(* IEC 61131-3 sources: AXOpen/src/components.zebra.vision/app/SystemConstants, 2 files *)

(* ---- plc_line_IoAddresses.st ---- *)
CONFIGURATION IoAddresses
    VAR_GLOBAL

        // Module EA3600/Data88Bin6Bout
        EA3600_Data88Bin6Bout_Input AT %IB0 : EA3600_Data88Bin6Bout_Input_Layout;
        EA3600_Data88Bin6Bout_Output AT %QB0 : EA3600_Data88Bin6Bout_Output_Layout;
    END_VAR
END_CONFIGURATION

TYPE
    EA3600_Data88Bin6Bout_Input_Layout : STRUCT
        Signals_0 AT %B0 : ARRAY[0..703] OF BOOL;
    END_STRUCT;
END_TYPE

TYPE
    EA3600_Data88Bin6Bout_Output_Layout : STRUCT
        Signals_1_0 AT %X0.0 : BOOL;
        Signals_1_1 AT %X0.1 : BOOL;
        Signals_1_2 AT %X0.2 : BOOL;
        Signals_1_3 AT %X0.3 : BOOL;
        Signals_1_4 AT %X0.4 : BOOL;
        Signals_1_5 AT %X0.5 : BOOL;
        Signals_1_6 AT %X0.6 : BOOL;
        Signals_1_7 AT %X0.7 : BOOL;
        Signals_1_8 AT %X1.0 : BOOL;
        Signals_1_9 AT %X1.1 : BOOL;
        Signals_1_10 AT %X1.2 : BOOL;
        Signals_1_11 AT %X1.3 : BOOL;
        Signals_1_12 AT %X1.4 : BOOL;
        Signals_1_13 AT %X1.5 : BOOL;
        Signals_1_14 AT %X1.6 : BOOL;
        Signals_1_15 AT %X1.7 : BOOL;
        Signals_1_16 AT %X2.0 : BOOL;
        Signals_1_17 AT %X2.1 : BOOL;
        Signals_1_18 AT %X2.2 : BOOL;
        Signals_1_19 AT %X2.3 : BOOL;
        Signals_1_20 AT %X2.4 : BOOL;
        Signals_1_21 AT %X2.5 : BOOL;
        Signals_1_22 AT %X2.6 : BOOL;
        Signals_1_23 AT %X2.7 : BOOL;
        Signals_1_24 AT %X3.0 : BOOL;
        Signals_1_25 AT %X3.1 : BOOL;
        Signals_1_26 AT %X3.2 : BOOL;
        Signals_1_27 AT %X3.3 : BOOL;
        Signals_1_28 AT %X3.4 : BOOL;
        Signals_1_29 AT %X3.5 : BOOL;
        Signals_1_30 AT %X3.6 : BOOL;
        Signals_1_31 AT %X3.7 : BOOL;
        Signals_1_32 AT %X4.0 : BOOL;
        Signals_1_33 AT %X4.1 : BOOL;
        Signals_1_34 AT %X4.2 : BOOL;
        Signals_1_35 AT %X4.3 : BOOL;
        Signals_1_36 AT %X4.4 : BOOL;
        Signals_1_37 AT %X4.5 : BOOL;
        Signals_1_38 AT %X4.6 : BOOL;
        Signals_1_39 AT %X4.7 : BOOL;
        Signals_1_40 AT %X5.0 : BOOL;
        Signals_1_41 AT %X5.1 : BOOL;
        Signals_1_42 AT %X5.2 : BOOL;
        Signals_1_43 AT %X5.3 : BOOL;
        Signals_1_44 AT %X5.4 : BOOL;
        Signals_1_45 AT %X5.5 : BOOL;
        Signals_1_46 AT %X5.6 : BOOL;
        Signals_1_47 AT %X5.7 : BOOL;
    END_STRUCT;
END_TYPE

(* ---- plc_line_HwIdentifiers.st ---- *)
CONFIGURATION HardwareIDs
    VAR_GLOBAL CONSTANT
        plc_line_HwID : UINT := UINT#32;
        plc_line_Rail_0_HwID : UINT := UINT#264;
        plc_line_plc_line_HwID : UINT := UINT#48;
        plc_line_plc_line_CPU_display_1_HwID : UINT := UINT#54;
        plc_line_plc_line_Card_reader_writer_1_HwID : UINT := UINT#51;
        plc_line_plc_line_OPC_UA_1_HwID : UINT := UINT#117;
        plc_line_plc_line_PROFINET_interface_1_HwID : UINT := UINT#64;
        plc_line_plc_line_PROFINET_interface_1_Port_1_HwID : UINT := UINT#65;
        plc_line_plc_line_PROFINET_interface_1_Port_2_HwID : UINT := UINT#66;
        plc_line_plc_line_PROFINET_interface_2_HwID : UINT := UINT#72;
        plc_line_plc_line_PROFINET_interface_2_Port_3_HwID : UINT := UINT#73;
        plc_line_plc_line_PROFINET_interface_2_Port_4_HwID : UINT := UINT#74;
        plc_line_plc_line_PROFINET_interface_GBIT_3_HwID : UINT := UINT#120;
        plc_line_plc_line_PROFINET_interface_GBIT_3_Port_5_HwID : UINT := UINT#121;
        plc_line_plc_line_Virtual_communication_interface_HwID : UINT := UINT#135;
        profinet_plc_line_HwID : UINT := UINT#256;
        zebra_HwID : UINT := UINT#258;
        zebra_Data88Bin6Bout_Data_and_Transfer_Control_v2_HwID : UINT := UINT#262;
        zebra_Rack_HwID : UINT := UINT#260;
        zebra_zebra_HwID : UINT := UINT#261;
        zebra_zebra_EA3600_PIO_Interface_HwID : UINT := UINT#263;
        zebra_zebra_Interface_HwID : UINT := UINT#257;
        zebra_zebra_Interface_Port_1_HwID : UINT := UINT#259;

    END_VAR
END_CONFIGURATION
